ADAPTER ADP_PRODUCTION_TOKEN (* Adapter Interface *)
  (* Standard: 61499-1 *)
  (* Version 0.0, 12/17/2022, Dmitrii, Flexbridge AB *)
  PACKAGE UAO.Hackathon;
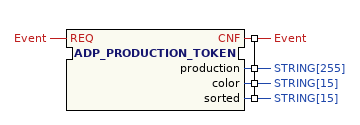
  EVENT_INPUT
    REQ; (* Request from Socket *)
  END_EVENT
  EVENT_OUTPUT
    CNF WITH production, sorted, color; (* Confirmation from Plug *)
  END_EVENT
  VAR_OUTPUT
    production : STRING[255]; (* Request Data from Socket *)
    color : STRING[15]; (* Confirmation Data from Plug *)
    sorted : STRING[15]; (* Indication Data from Plug *)
  END_VAR
  SERVICE SOCKET/PLUG
    SEQUENCE request_confirm
      SOCKET.REQ(production) -> PLUG.REQ(production);
      PLUG.CNF(color) -> SOCKET.CNF(color);
    END_SEQUENCE
    SEQUENCE indication_response
      PLUG.IND(sorted) -> SOCKET.IND(sorted);
      SOCKET.RSP(RSPD) -> PLUG.RSP(RSPD);
    END_SEQUENCE
  END_SERVICE
END_ADAPTER
